(* CODESYS project E1.project

Project tree, tasks and I/O mapping:
  Device : CODESYS Control Win V3, 3S - Smart Software Solutions GmbH, order no. 305021, version 3.5.4.40
    application Application
      libraries: Standard, * (System)
      task MainTask (cyclic, interval t#20ms, priority 1) calls PLC_PRG
      program PLC_PRG [LD]
*)

// Device/Application/PLC_PRG
PROGRAM PLC_PRG
VAR
	I0: BOOL;
	Q4: BOOL;
	In1: BOOL;
	In2: BOOL;
	O1: BOOL;
	O2: BOOL;
	BB1: RS;
	BB2: SR;
END_VAR

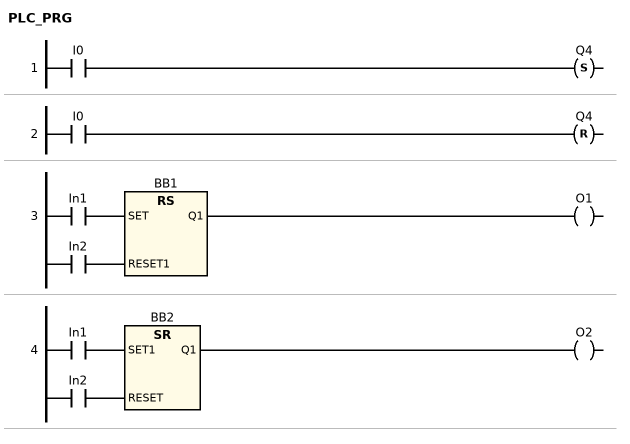
// NETWORK 1
Q4 S= I0;

// NETWORK 2
Q4 R= I0;

// NETWORK 3
BB1(SET := In1, RESET1 := In2); // RS
O1 := BB1.Q1;

// NETWORK 4
BB2(SET1 := In1, RESET := In2); // SR
O2 := BB2.Q1;

END_PROGRAM
